Omron CX-Programmer project NewProject (CX-Programmer 9.54)

# PLC Automation_project_Station2: CJ1M CPU11

## Global symbols (name address type ; comment)
0.00 BOOL  ; Start_PB
0.01 BOOL  ; Stop_PB
0.02 BOOL  ; Reset_PB
0.03 BOOL  ; Emergency_PB
0.04 BOOL  ; Pusher 3 Front Limit
0.05 BOOL  ; Machining_Busy
0.06 BOOL  ; Machining_Error
0.07 BOOL  ; Machining_Opened
0.08 BOOL  ; Machining_Progress
0.09 BOOL  ; Vision 3
0.10 BOOL  ; Diff_Sensor3
0.11 BOOL  ; Diff_Sensor_Base
0.12 BOOL  ; Diff_Sensor_Lid
0.13 BOOL  ; Base Positioner Up Limit
0.14 BOOL  ; Base Positioner Limit
0.15 BOOL  ; Lid Positioner Limit
1.00 BOOL  ; Blue Base Conveyor
1.01 BOOL  ; Machining_Start
1.04 BOOL  ; Pusher 3
1.05 BOOL  ; Base Positioner Up
1.06 BOOL  ; Pick_Place_X
1.07 BOOL  ; Pick_Place_Z
1.08 BOOL  ; Lid Positioner Clamp
1.09 BOOL  ; Base Positioner Clamp
1.10 BOOL  ; Roller Stopper 3
1.11 BOOL  ; Green Lid Conveyor
1.12 BOOL  ; Pick_Place_Grab
1.13 BOOL  ; Start_Light
1.14 BOOL  ; Stop_Light
1.15 BOOL  ; Reset_Light
D10 CHANNEL  ; Assembly Counting
D100 CHANNEL  ; Step
D11 CHANNEL  ; Reject Counting
D12 CHANNEL  ; Lid Counting
D13 CHANNEL  ; Base Counting
W10.00 BOOL  ; Pusher Control
W10.01 BOOL  ; Roller Stopper Control
W10.02 BOOL  ; Pusher Control
W10.03 BOOL  ; Painted Emitter Control
W10.04 BOOL  ; Reset Counting
W11.00 BOOL  ; Counting_Control_Painted
W11.01 BOOL  ; Counting_Control_Reject
W1.00 BOOL  ; Status
W1.01 BOOL  ; Emergency_Status
W20.00 BOOL  ; Machining_Busy_Status
W20.01 BOOL  ; Machining_Error_Status
W20.02 BOOL  ; Machining_Opened_Status
W20.03 BOOL  ; Machining_Progress_Status
W30.00 BOOL  ; Grab_Control
W30.01 BOOL  ; Pick_Place_Z_Control
W30.02 BOOL  ; Pick_Place_X_Control
W30.03 BOOL  ; Base Positioner Up Control

## Program NewProgram1 (cyclic task 0)

### Section Init

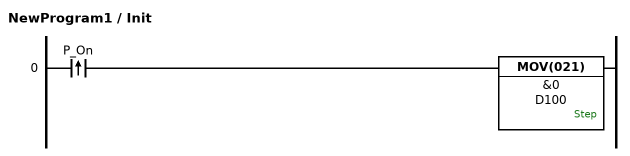
; rung 0
@LD P_On
MOV(021) &0 D100  ; Step

### Section Station3

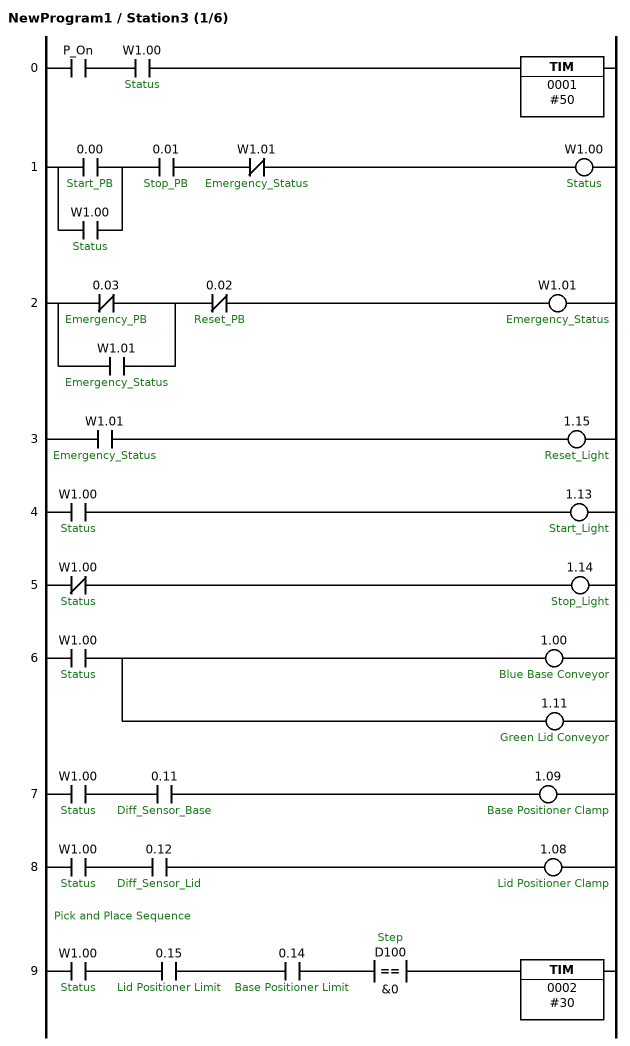
; rung 0
LD P_On
AND W1.00  ; Status
TIM 0001 #50
; rung 1
LD 0.00  ; Start_PB
OR W1.00  ; Status
AND 0.01  ; Stop_PB
ANDNOT W1.01  ; Emergency_Status
OUT W1.00  ; Status
; rung 2
LDNOT 0.03  ; Emergency_PB
OR W1.01  ; Emergency_Status
ANDNOT 0.02  ; Reset_PB
OUT W1.01  ; Emergency_Status
; rung 3
LD W1.01  ; Emergency_Status
OUT 1.15  ; Reset_Light
; rung 4
LD W1.00  ; Status
OUT 1.13  ; Start_Light
; rung 5
LDNOT W1.00  ; Status
OUT 1.14  ; Stop_Light
; rung 6
LD W1.00  ; Status
OUT 1.00  ; Blue Base Conveyor
OUT 1.11  ; Green Lid Conveyor
; rung 7
LD W1.00  ; Status
AND 0.11  ; Diff_Sensor_Base
OUT 1.09  ; Base Positioner Clamp
; rung 8
LD W1.00  ; Status
AND 0.12  ; Diff_Sensor_Lid
OUT 1.08  ; Lid Positioner Clamp
; rung 9: Pick and Place Sequence
LD W1.00  ; Status
AND 0.15  ; Lid Positioner Limit
AND 0.14  ; Base Positioner Limit
AND=(300) D100 &0  ; Step
TIM 0002 #30

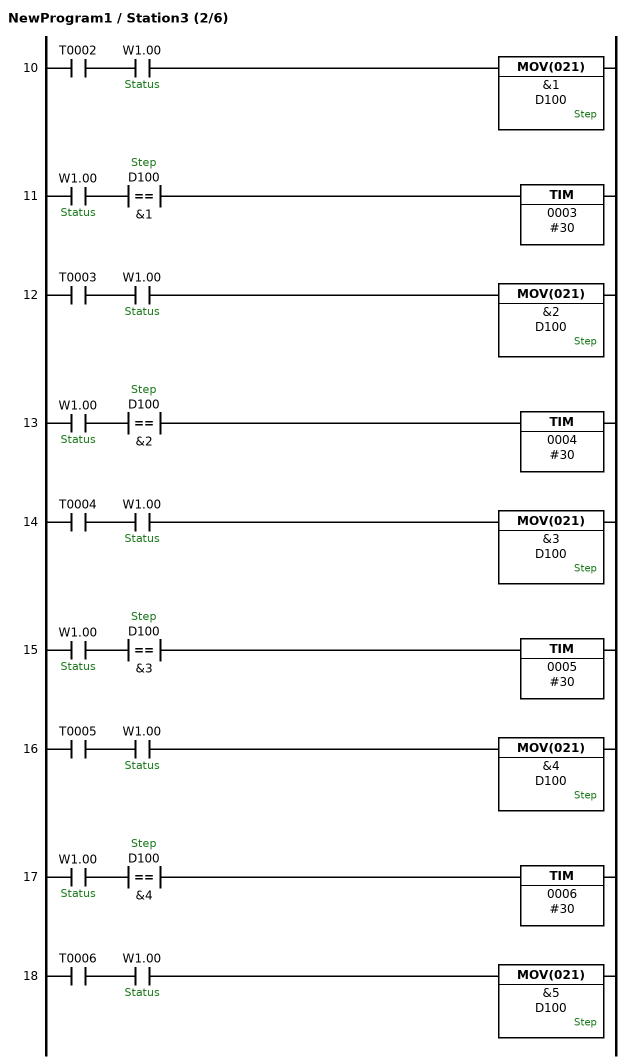
; rung 10
LD T0002
AND W1.00  ; Status
MOV(021) &1 D100  ; Step
; rung 11
LD W1.00  ; Status
AND=(300) D100 &1  ; Step
TIM 0003 #30
; rung 12
LD T0003
AND W1.00  ; Status
MOV(021) &2 D100  ; Step
; rung 13
LD W1.00  ; Status
AND=(300) D100 &2  ; Step
TIM 0004 #30
; rung 14
LD T0004
AND W1.00  ; Status
MOV(021) &3 D100  ; Step
; rung 15
LD W1.00  ; Status
AND=(300) D100 &3  ; Step
TIM 0005 #30
; rung 16
LD T0005
AND W1.00  ; Status
MOV(021) &4 D100  ; Step
; rung 17
LD W1.00  ; Status
AND=(300) D100 &4  ; Step
TIM 0006 #30
; rung 18
LD T0006
AND W1.00  ; Status
MOV(021) &5 D100  ; Step

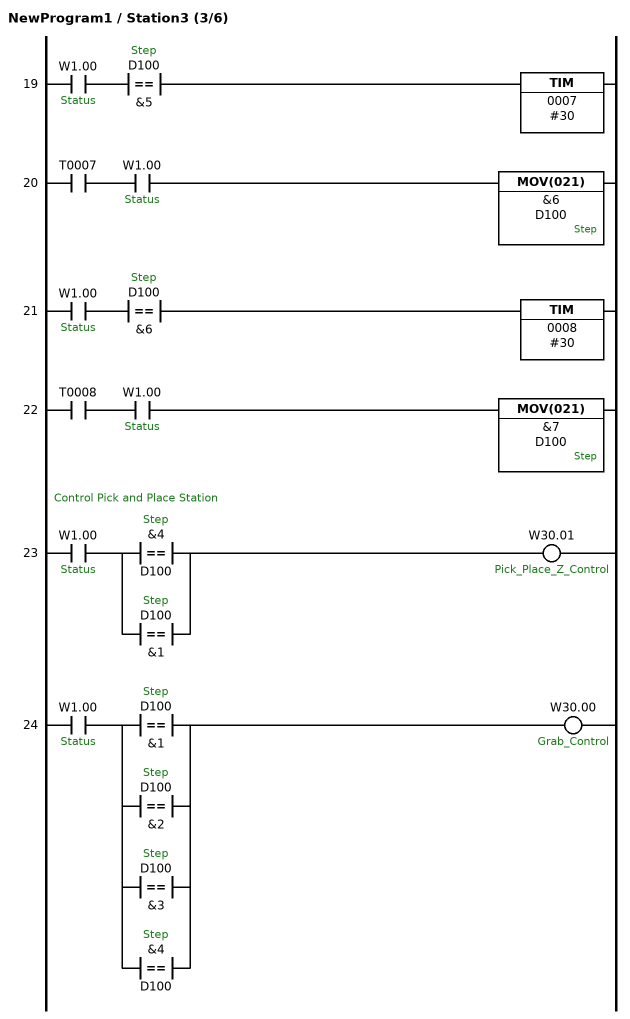
; rung 19
LD W1.00  ; Status
AND=(300) D100 &5  ; Step
TIM 0007 #30
; rung 20
LD T0007
AND W1.00  ; Status
MOV(021) &6 D100  ; Step
; rung 21
LD W1.00  ; Status
AND=(300) D100 &6  ; Step
TIM 0008 #30
; rung 22
LD T0008
AND W1.00  ; Status
MOV(021) &7 D100  ; Step
; rung 23: Control Pick and Place Station
LD W1.00  ; Status
LD=(300) &4 D100  ; Step
OR=(300) D100 &1  ; Step
ANDLD
OUT W30.01  ; Pick_Place_Z_Control
; rung 24
LD W1.00  ; Status
LD=(300) D100 &1  ; Step
OR=(300) D100 &2  ; Step
OR=(300) D100 &3  ; Step
OR=(300) &4 D100  ; Step
ANDLD
OUT W30.00  ; Grab_Control

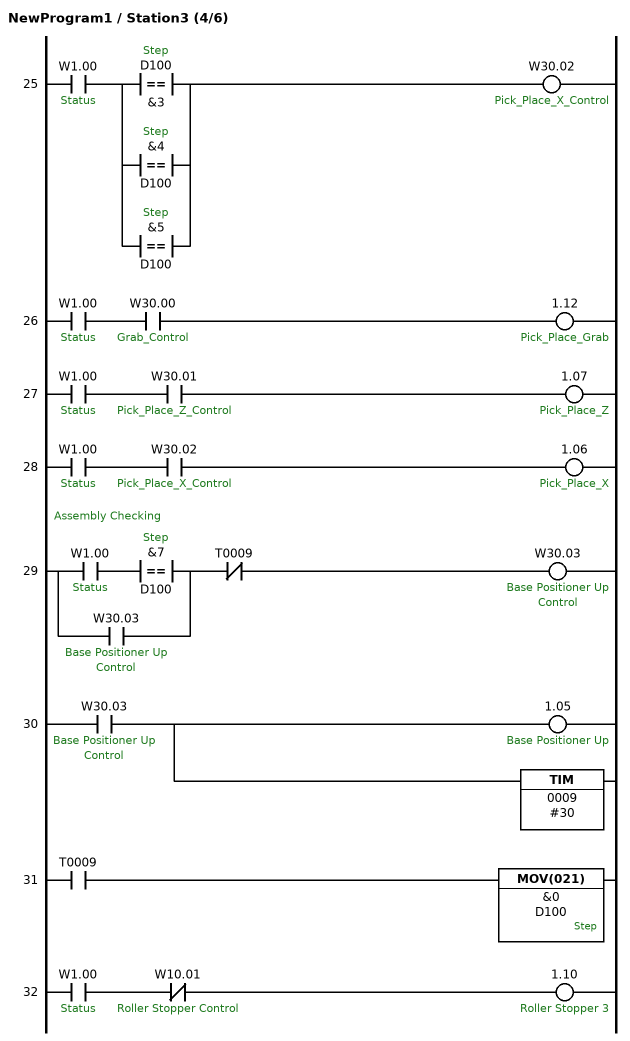
; rung 25
LD W1.00  ; Status
LD=(300) D100 &3  ; Step
OR=(300) &4 D100  ; Step
OR=(300) &5 D100  ; Step
ANDLD
OUT W30.02  ; Pick_Place_X_Control
; rung 26
LD W1.00  ; Status
AND W30.00  ; Grab_Control
OUT 1.12  ; Pick_Place_Grab
; rung 27
LD W1.00  ; Status
AND W30.01  ; Pick_Place_Z_Control
OUT 1.07  ; Pick_Place_Z
; rung 28
LD W1.00  ; Status
AND W30.02  ; Pick_Place_X_Control
OUT 1.06  ; Pick_Place_X
; rung 29: Assembly Checking
LD W1.00  ; Status
AND=(300) &7 D100  ; Step
OR W30.03  ; Base Positioner Up Control
ANDNOT T0009
OUT W30.03  ; Base Positioner Up Control
; rung 30
LD W30.03  ; Base Positioner Up Control
OUT 1.05  ; Base Positioner Up
TIM 0009 #30
; rung 31
LD T0009
MOV(021) &0 D100  ; Step
; rung 32
LD W1.00  ; Status
ANDNOT W10.01  ; Roller Stopper Control
OUT 1.10  ; Roller Stopper 3

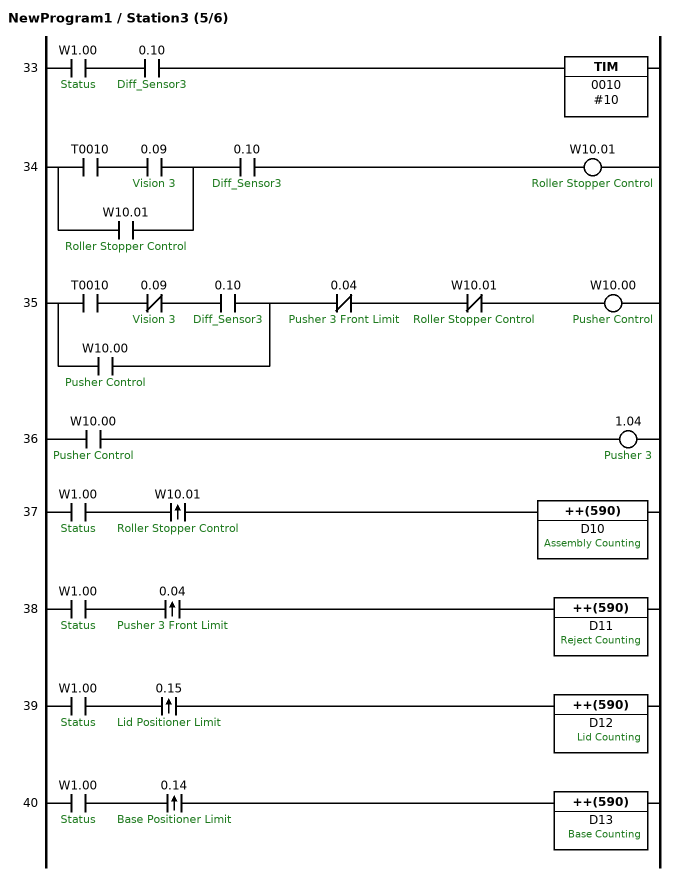
; rung 33
LD W1.00  ; Status
AND 0.10  ; Diff_Sensor3
TIM 0010 #10
; rung 34
LD T0010
AND 0.09  ; Vision 3
OR W10.01  ; Roller Stopper Control
AND 0.10  ; Diff_Sensor3
OUT W10.01  ; Roller Stopper Control
; rung 35
LD T0010
ANDNOT 0.09  ; Vision 3
AND 0.10  ; Diff_Sensor3
OR W10.00  ; Pusher Control
ANDNOT 0.04  ; Pusher 3 Front Limit
ANDNOT W10.01  ; Roller Stopper Control
OUT W10.00  ; Pusher Control
; rung 36
LD W10.00  ; Pusher Control
OUT 1.04  ; Pusher 3
; rung 37
LD W1.00  ; Status
@AND W10.01  ; Roller Stopper Control
++(590) D10  ; Assembly Counting
; rung 38
LD W1.00  ; Status
@AND 0.04  ; Pusher 3 Front Limit
++(590) D11  ; Reject Counting
; rung 39
LD W1.00  ; Status
@AND 0.15  ; Lid Positioner Limit
++(590) D12  ; Lid Counting
; rung 40
LD W1.00  ; Status
@AND 0.14  ; Base Positioner Limit
++(590) D13  ; Base Counting

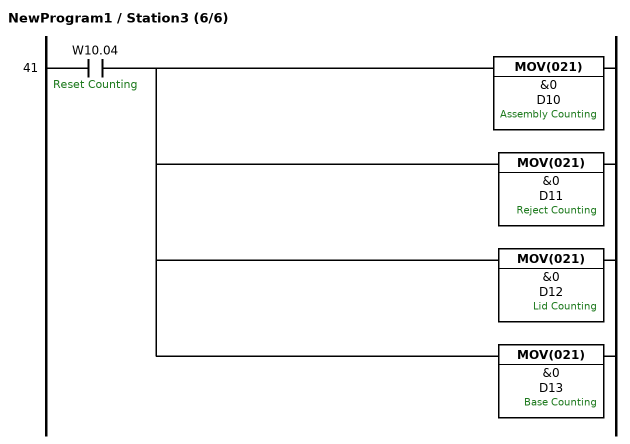
; rung 41
LD W10.04  ; Reset Counting
MOV(021) &0 D10  ; Assembly Counting
MOV(021) &0 D11  ; Reject Counting
MOV(021) &0 D12  ; Lid Counting
MOV(021) &0 D13  ; Base Counting

### Section Lid_Machining_Control

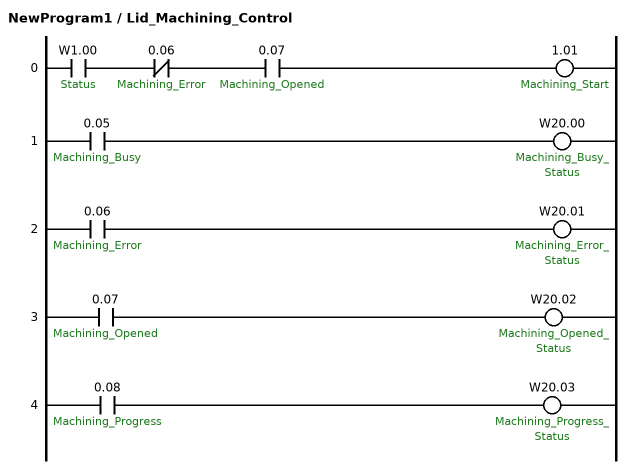
; rung 0
LD W1.00  ; Status
ANDNOT 0.06  ; Machining_Error
AND 0.07  ; Machining_Opened
OUT 1.01  ; Machining_Start
; rung 1
LD 0.05  ; Machining_Busy
OUT W20.00  ; Machining_Busy_Status
; rung 2
LD 0.06  ; Machining_Error
OUT W20.01  ; Machining_Error_Status
; rung 3
LD 0.07  ; Machining_Opened
OUT W20.02  ; Machining_Opened_Status
; rung 4
LD 0.08  ; Machining_Progress
OUT W20.03  ; Machining_Progress_Status

### Section END
; rung 0
END(001)